(* IEC 61131-3 sources: AXOpen/src/data/app/src/Examples, 4 files *)

(* ---- AxoDataDistributedExample.st ---- *)
USING AXOpen.Core;
USING AXOpen.Data;

NAMESPACE AxoDataDistributedExample

    //<ContextDeclaration>
    {S7.extern=ReadWrite}
    CLASS PUBLIC Context EXTENDS AXOpen.Core.AxoContext
        VAR PUBLIC
            //Controlled unit that needs to manipulate with data
            {#ix-set:AttributeName = "Unit 1"}
            ControlledUnit_1 : ControlledUnit;

            {#ix-set:AttributeName = "Unit 2"}
            ControlledUnit_2 : ControlledUnit;
        END_VAR

        METHOD OVERRIDE Main
            THIS.InitializeRootObject(ControlledUnit);
            ControlledUnit.Run();// run logic of controlled unit
        END_METHOD
    END_CLASS
    //</ContextDeclaration>

    {S7.extern=ReadWrite}
    CLASS PUBLIC SharedHeader_Manager
        EXTENDS AXOpen.Data.AxoDataExchange
        VAR PUBLIC
            {#ix-generic:TOnline}
            {#ix-generic:TPlain as POCO}
            {#ix-attr:[AXOpen.Data.AxoDataEntityAttribute]}
            {#ix-attr:[Container(Layout.Stack)]}
            {#ix-set:AttributeName = "Shared Header"}
            Set : SharedHeader_Data;
        END_VAR
    END_CLASS

    {S7.extern=ReadWrite}
    CLASS PUBLIC SharedHeader_Data
        EXTENDS AXOpen.Data.AxoDataEntity
        VAR PUBLIC
            HeaderPartialName : STRING;
            HeaderIndex : INT;
            HeaderGlogalPass : BOOL;
        END_VAR
    END_CLASS

    {S7.extern=ReadWrite}
    CLASS PUBLIC StationData_Manager
        EXTENDS AXOpen.Data.AxoDataExchange
        VAR PUBLIC
            {#ix-generic:TOnline}
            {#ix-generic:TPlain as POCO}
            {#ix-attr:[AXOpen.Data.AxoDataEntityAttribute]}
            {#ix-attr:[Container(Layout.Stack)]}
            {#ix-set:AttributeName = "Station"}
            Set : Station_Data;
        END_VAR
    END_CLASS

    {S7.extern=ReadWrite}
    CLASS PUBLIC Station_Data EXTENDS AXOpen.Data.AxoDataEntity
        VAR PUBLIC
            StationName : STRING;
            StaionOperation : INT;
            StationPass : BOOL;
        END_VAR
    END_CLASS

     {S7.extern=ReadWrite}
     CLASS PUBLIC ManagerUsage
        VAR PUBLIC
            _id : STRING;
            _create : BOOL;
            _update : BOOL;
            _read : BOOL;
            _delete : BOOL;
        END_VAR

        METHOD PUBLIC Use
            VAR_IN_OUT
                DataManager : AXOpen.Data.AxoDataExchange;
            END_VAR
            IF(_create) THEN
                IF(DataManager.Create(_id).IsDone()) THEN
                    _create := FALSE;
                END_IF;
            END_IF;

            IF(_read) THEN
                IF(DataManager.Read(_id).IsDone()) THEN
                    _read := FALSE;
                END_IF;
            END_IF;

            IF(_update) THEN
                IF(DataManager.Update(_id).IsDone()) THEN
                    _update := FALSE;
                END_IF;
            END_IF;

            IF(_delete) THEN
                IF(DataManager.Delete(_id).IsDone()) THEN
                    _delete := FALSE;
                END_IF;
            END_IF;
        END_METHOD
    END_CLASS

    {S7.extern=ReadWrite}
    CLASS PUBLIC ControlledUnit EXTENDS AXOpen.Core.AxoObject
        VAR PUBLIC

            //<UseDistributedDataAttribute>
            {#ix-attr:[AXOpen.Data.DistributedDataAttribute("default", "headers")]}
            EntityHeader : SharedHeader_Manager;
            {#ix-attr:[AXOpen.Data.DistributedDataAttribute("default", "headers")]}
            ProcessData : StationData_Manager;
            //</UseDistributedDataAttribute>

            HeaderUsage : ManagerUsage;
            ProcessUsage : ManagerUsage;

            //Automatic sequence. Contains logic for automatic operations of this unit.
            AutomatSequence : AutomatSequence;
        END_VAR

        METHOD PUBLIC Run
            SUPER.Run(THIS); //??
            THIS.EntityHeader.Run(THIS)
            THIS.ProcessData.Run(THIS)

            HeaderUsage.Run(THIS);
            ProcessUsage.Run(THIS);

            THIS.Execute();
        END_METHOD

        METHOD PRIVATE Execute
            ProcessData^.Run(THIS); // cyclic call of AxoProcessDataManager
            AutomatSequence.Run(THIS, ^ProcessData);
        END_METHOD
    END_CLASS

    //<Run>
    {S7.extern=ReadWrite}
    CLASS PUBLIC AutomatSequence EXTENDS AXOpen.Core.AxoSequencerContainer
        VAR PRIVATE
            // private reference is used in Main()
            HeaderData : REF_TO SharedHeader_Manager;
            ProcessData : REF_TO StationData_Manager;
        END_VAR

        METHOD INTERNAL Run
            VAR_INPUT
                _parent : IAxoObject;
                _processData : REF_TO StationData_Manager;
                _headerData : REF_TO SharedHeader_Manager;
            END_VAR

            ProcessData := _processData;
            HeaderData := _headerData;
        END_METHOD

        METHOD OVERRIDE Main
            ;//cyclic logic
        END_METHOD
    END_CLASS
    //</Run>

END_NAMESPACE

(* ---- AxoDataExchangeExample.st ---- *)
USING AXOpen.Core;
USING AXOpen;
using AXOpen.Data;

NAMESPACE AxoDataExchangeExample

    //<ContextDeclaration>
    {S7.extern=ReadWrite}
    CLASS PUBLIC Context EXTENDS AXOpen.Core.AxoContext
        VAR PUBLIC
            //Controlled unit that needs to manipulate with data
            ControlledUnit : ControlledUnit;
            //DataManager instance
            DataManager  : AxoProcessDataManager;

            //Testing usage of the manager
            ManagerUsage : ManagerUsage;
        END_VAR

        METHOD OVERRIDE Main

            // DataManager.Run(THIS); - is called iside of controlle unit
            THIS.InitializeRootObject(ControlledUnit);
            ControlledUnit.ProcessData := REF(DataManager);//Set REF to DataManager (reason depth of data structure)
            ControlledUnit.Run();// run logic of controlled unit

            ManagerUsage.Use(DataManager);
        END_METHOD
    END_CLASS
    //</ContextDeclaration>

    //<AxoProcessDataManagerDeclaration>
    {S7.extern=ReadWrite}
    CLASS PUBLIC AxoProcessDataManager EXTENDS AXOpen.Data.AxoDataExchange
        VAR PUBLIC
            {#ix-generic:TOnline}
            {#ix-generic:TPlain as POCO}
            {#ix-attr:[AXOpen.Data.AxoDataEntityAttribute]}
            Set : AxoProcessData; // <- Manager will operate on this member.
        END_VAR
    END_CLASS
    //</AxoProcessDataManagerDeclaration>

    //<AxoProcessDataDeclaration>
    {S7.extern=ReadWrite}
    CLASS PUBLIC AxoProcessData EXTENDS AXOpen.Data.AxoDataEntity
        VAR PUBLIC
            {#ix-set:AttributeName = "Some string"}
            SomeString : STRING;
            {#ix-set:AttributeName = "Some int"}
            SomeInt : INT;

            AllPrimitives : BasePrimitives;
        END_VAR
    END_CLASS
    //</AxoProcessDataDeclaration>

    //<Usage>
    {S7.extern=ReadWrite}
    CLASS PUBLIC ManagerUsage
        VAR PUBLIC
            _id : STRING;
            _create : BOOL;
            _update : BOOL;
            _read : BOOL;
            _delete : BOOL;
        END_VAR

        METHOD PUBLIC Use
            VAR_IN_OUT
                DataManager : AxoProcessDataManager;
            END_VAR
            IF(_create) THEN
                IF(DataManager.Create(_id).IsDone()) THEN
                    _create := FALSE;
                END_IF;
            END_IF;

            IF(_read) THEN
                IF(DataManager.Read(_id).IsDone()) THEN
                    _read := FALSE;
                END_IF;
            END_IF;

            IF(_update) THEN
                IF(DataManager.Update(_id).IsDone()) THEN
                    _update := FALSE;
                END_IF;
            END_IF;

            IF(_delete) THEN
                IF(DataManager.Delete(_id).IsDone()) THEN
                    _delete := FALSE;
                END_IF;
            END_IF;
        END_METHOD
    END_CLASS
    //</Usage>

    //<Execute>
    {S7.extern=ReadWrite}
    CLASS PUBLIC ControlledUnit EXTENDS AXOpen.Core.AxoObject
        VAR PUBLIC
            //Reference to ProcessDataManager
            ProcessData : REF_TO AxoProcessDataManager;
            //Automatic sequence. Contains logic for automatic operations of this unit.
            AutomatSequence : AutomatSequence;
        END_VAR

        METHOD PUBLIC Run
            SUPER.Run(THIS); //??
            THIS.Execute();
        END_METHOD

        METHOD PRIVATE Execute
            ProcessData^.Run(THIS); // cyclic call of AxoProcessDataManager
            AutomatSequence.Run(THIS, ProcessData);
        END_METHOD
    END_CLASS
    //</Execute>

    //<Run>
    {S7.extern=ReadWrite}
    CLASS PUBLIC AutomatSequence EXTENDS AXOpen.Core.AxoSequencerContainer
        VAR PRIVATE
            // private reference is used in Main()
            ProcessData : REF_TO AxoProcessDataManager;
        END_VAR

        METHOD INTERNAL Run
            VAR_INPUT
                _parent : IAxoObject;
                _processData : REF_TO AxoProcessDataManager;
            END_VAR

            ProcessData := _processData;
        END_METHOD

        METHOD OVERRIDE Main
            ;//cyclic logic
        END_METHOD
    END_CLASS
    //</Run>

    {S7.extern=ReadWrite}
    CLASS PUBLIC BasePrimitives //27 vars
        VAR PUBLIC
            vBOOL           :       BOOL	      ;
            vBYTE           :       BYTE	      ;
            vWORD           :       WORD	      ;
            vDWORD          :       DWORD	      ;
            vLWORD	        :       LWORD	      ;
            vSINT           :       SINT	      ;
            vINT	        :       INT           ;
            vDINT	        :       DINT	      ;
            vLINT	        :       LINT	      ;
            vUSINT	        :       USINT	      ;
            vUINT	        :       UINT	      ;
            vUDINT	        :       UDINT	      ;
            vULINT	        :       ULINT	      ;
            vREAL	        :       REAL	      ;
            vLREAL	        :       LREAL	      ;
            vTIME	        :       TIME	      ;
            vLTIME	        :       LTIME	      ;
            vDATE	        :       DATE	      ;
            vLDATE	        :       LDATE	      ;
            vTIME_OF_DAY	:       TIME_OF_DAY   ;
            vLTIME_OF_DAY	:       LTIME_OF_DAY  ;
            vDATE_AND_TIME  :      DATE_AND_TIME  ;
            vLDATE_AND_TIME :      LDATE_AND_TIME ;
            vCHAR	        :       CHAR	      ;
            vWCHAR	        :       WCHAR	      ;
            vSTRING         :       STRING	      ;
            vWSTRING        :       WSTRING	      ;
        END_VAR
    END_CLASS

END_NAMESPACE

(* ---- AxoDataFragmentExchangeExample.st ---- *)
USING AXOpen.Core;
USING AXOpen.Data;

NAMESPACE AxoDataFramentsExchangeExample

    //<ContextDeclaration>
    {S7.extern=ReadWrite}
    CLASS PUBLIC Context EXTENDS AXOpen.Core.AxoContext
        VAR PUBLIC
            //Controlled unit that needs to manipulate with data
            ControlledUnit : ControlledUnit;
            //DataManager instance
            DataManager  : AxoProcessDataManager;

            //Testing usage of the manager
            ManagerUsage : ManagerUsage;
        END_VAR

        METHOD OVERRIDE Main

            // DataManager.Run(THIS); - is called iside of controlle unit
            ControlledUnit.ProcessData := REF(DataManager);//Set REF to DataManager (reason depth of data structure)
            ControlledUnit.Run(THIS);// run logic of controlled unit

            ManagerUsage.Use(DataManager);
        END_METHOD
    END_CLASS
    //</ContextDeclaration>

    //<AxoProcessDataManagerDeclaration>
    {S7.extern=ReadWrite}
    CLASS PUBLIC AxoProcessDataManager
        EXTENDS AXOpen.Data.AxoDataFragmentExchange
        VAR PUBLIC
            {#ix-attr:[AXOpen.Data.AxoDataFragmentAttribute]}
            SharedHeader : SharedDataHeaderManager;
            {#ix-attr:[AXOpen.Data.AxoDataFragmentAttribute]}
            Station_1 : Station_1_ProcessDataManager;
        END_VAR
    END_CLASS
    //</AxoProcessDataManagerDeclaration>

    {S7.extern=ReadWrite}
    CLASS PUBLIC SharedDataHeaderManager
        EXTENDS AXOpen.Data.AxoDataExchange
        VAR PUBLIC
            {#ix-generic:TOnline}
            {#ix-generic:TPlain as POCO}
            {#ix-attr:[AXOpen.Data.AxoDataEntityAttribute]}
            {#ix-attr:[Container(Layout.Stack)]}
            {#ix-set:AttributeName = "Shared Header"}
            Set : SharedDataHeaderData;
        END_VAR
    END_CLASS

    {S7.extern=ReadWrite}
    CLASS PUBLIC SharedDataHeaderData
        EXTENDS AXOpen.Data.AxoDataEntity
        VAR PUBLIC
            {#ix-set:AttributeName = "Some string"}
            SomeString : STRING;
            {#ix-set:AttributeName = "Some int"}
            SomeInt : INT;
            {#ix-set:AttributeName = "Some bool"}
            SomeBool : BOOL;
        END_VAR
    END_CLASS

    {S7.extern=ReadWrite}
    CLASS PUBLIC Station_1_ProcessDataManager
        EXTENDS AXOpen.Data.AxoDataExchange
        VAR PUBLIC
            {#ix-generic:TOnline}
            {#ix-generic:TPlain as POCO}
            {#ix-attr:[AXOpen.Data.AxoDataEntityAttribute]}
            {#ix-attr:[Container(Layout.Stack)]}
            {#ix-set:AttributeName = "Station 1"}
            Set : Station_1_Data;
        END_VAR
    END_CLASS

    {S7.extern=ReadWrite}
    CLASS PUBLIC Station_1_Data EXTENDS AXOpen.Data.AxoDataEntity
        VAR PUBLIC
            {#ix-set:AttributeName = "Some string st"}
            SomeString : STRING;
            {#ix-set:AttributeName = "Some int st"}
            SomeInt : INT;
            {#ix-set:AttributeName = "Some bool st"}
            SomeBool : BOOL;
        END_VAR
    END_CLASS

     //<Usage>
     {S7.extern=ReadWrite}
     CLASS PUBLIC ManagerUsage
        VAR PUBLIC
            _id : STRING;
            _create : BOOL;
            _update : BOOL;
            _read : BOOL;
            _delete : BOOL;
        END_VAR

        METHOD PUBLIC Use
            VAR_IN_OUT
                DataManager : AxoProcessDataManager;
            END_VAR
            IF(_create) THEN
                IF(DataManager.Create(_id).IsDone()) THEN
                    _create := FALSE;
                END_IF;
            END_IF;

            IF(_read) THEN
                IF(DataManager.Read(_id).IsDone()) THEN
                    _read := FALSE;
                END_IF;
            END_IF;

            IF(_update) THEN
                IF(DataManager.Update(_id).IsDone()) THEN
                    _update := FALSE;
                END_IF;
            END_IF;

            IF(_delete) THEN
                IF(DataManager.Delete(_id).IsDone()) THEN
                    _delete := FALSE;
                END_IF;
            END_IF;
        END_METHOD
    END_CLASS
    //</Usage>

    //<Execute>
    {S7.extern=ReadWrite}
    CLASS PUBLIC ControlledUnit EXTENDS AXOpen.Core.AxoObject
        VAR PUBLIC
            //Reference to ProcessDataManager
            ProcessData : REF_TO AxoProcessDataManager;
            //Automatic sequence. Contains logic for automatic operations of this unit.
            AutomatSequence : AutomatSequence;
        END_VAR

        METHOD PUBLIC Run
            VAR_INPUT
                _parent : IAxoContext;
            END_VAR
            THIS.Initialize(_parent);
            THIS.Execute();
        END_METHOD

        METHOD PRIVATE Execute
            ProcessData^.Run(THIS); // cyclic call of AxoProcessDataManager
            AutomatSequence.Run(THIS, ProcessData);
        END_METHOD
    END_CLASS
    //</Execute>

    //<Run>
    {S7.extern=ReadWrite}
    CLASS PUBLIC AutomatSequence EXTENDS AXOpen.Core.AxoSequencerContainer
        VAR PRIVATE
            // private reference is used in Main()
            ProcessData : REF_TO AxoProcessDataManager;
        END_VAR

        METHOD INTERNAL Run
            VAR_INPUT
                _parent : IAxoObject;
                _processData : REF_TO AxoProcessDataManager;
            END_VAR

            ProcessData := _processData;
        END_METHOD

        METHOD OVERRIDE Main
            ;//cyclic logic
        END_METHOD
    END_CLASS
    //</Run>

END_NAMESPACE

(* ---- AxoDataPersistentExchangeExample.st ---- *)
USING AXOpen.Core;
USING AXOpen;
using AXOpen.Data;

NAMESPACE AxoDataPersistentExchangeExample

    //<ContextDeclaration>
    {S7.extern=ReadWrite}
    CLASS PUBLIC Context EXTENDS AXOpen.Core.AxoContext
        VAR PUBLIC
            //persistent manager instance
            DataManager : AXOpen.Data.AxoDataPersistentExchange;
            //Testing usage of the manager
            ManagerUsage : ManagerUsage;
            // Object that propertie will be tracked by persistent manager
            PersistentRootObject : PersistentRootObject;
            _rootObject :   AxoObject;
        END_VAR

        METHOD OVERRIDE Main
            _rootObject.InitializeWithContext(THIS);
            DataManager.Run(_rootObject);
            ManagerUsage.Use(DataManager);
        END_METHOD
    END_CLASS
    //</ContextDeclaration>

    //<Usage>
    {S7.extern=ReadWrite}
    CLASS PUBLIC ManagerUsage EXTENDS AxOpen.Core.AxoObject
        VAR PUBLIC
            _persistentGroupId : STRING;
            _update : BOOL;
            _read : BOOL;
            _updateAll : BOOL;
            _readAll : BOOL;
            _exist : BOOL;
            _recordExist : BOOL;
        END_VAR

        METHOD PUBLIC Use
            VAR_IN_OUT
                DataManager : AXOpen.Data.AxoDataPersistentExchange;
            END_VAR

            IF(_read) THEN
                IF(DataManager.InvokeRead(THIS,_persistentGroupId)) THEN
                    ;
                END_IF;

                IF(DataManager.IsReadDone(THIS)) THEN
                    _read := FALSE;
                END_IF;
            END_IF;

            IF(_update) THEN
                IF(DataManager.InvokeUpdate(THIS,_persistentGroupId)) THEN
                   ;
                END_IF;

                IF(DataManager.IsUpdateDone(THIS)) THEN
                    _update := FALSE;
                END_IF;
            END_IF;

            IF(_readAll) THEN
                IF(DataManager.InvokeReadAll(THIS)) THEN
                   ;
                END_IF;
                IF(DataManager.IsReadAllDone(THIS)) THEN
                    _readAll := FALSE;
                END_IF;
            END_IF;

            IF(_updateAll) THEN
                IF(DataManager.InvokeUpdateAll(THIS)) THEN
                    ;
                END_IF;

                IF(DataManager.IsUpdateAllDone(THIS)) THEN
                    _updateAll := FALSE;
                END_IF;
            END_IF;

            IF(_exist) THEN
                IF(DataManager.InvokeEntityExist(THIS, _persistentGroupId)) THEN
                    ;
                END_IF;

                IF(DataManager.IsEntityExistDone(THIS)) THEN
                    _exist := FALSE;
                    _recordExist := DataManager.Operation._exist;
                END_IF;
            END_IF;
        END_METHOD
    END_CLASS
    //</ConcurrentUsage>

    //<PersistentAttribute>
    {S7.extern=ReadWrite}
    CLASS PUBLIC PersistentRootObject
        VAR PUBLIC
            NotPersistentVariable : BOOL;

            {#ix-attr:[Persistent()]}
            {#ix-set:AttributeName = "PersistentVariable_1 (in default pg.))"}
            PersistentVariable_1 : INT; // will be saved to 'default' persistent group

            {#ix-attr:[Persistent("default","1")]} // will be saved to 'default' and '1' persistent group
            {#ix-set:AttributeName = "PersistentVariable_2 (in default & 1 pg.)"}
            PersistentVariable_2 : INT;

            {#ix-attr:[Container(Layout.Stack)]}
            {#ix-attr:[Group(GroupLayout.GroupBox)]}
            {#ix-set:AttributeName = "PropertyWithPersistentMember"}
            PropertyWithPersistentMember : ObjectWithPersistentMember;
        END_VAR
    END_CLASS

    {S7.extern=ReadWrite}
    CLASS PUBLIC ObjectWithPersistentMember
        VAR PUBLIC
            NotPersistentVariable : INT;

            {#ix-attr:[Persistent("2")]}
            {#ix-attr:[Container(Layout.Stack)]}
            {#ix-attr:[Group(GroupLayout.GroupBox)]}
            {#ix-set:AttributeName = "InitializedPrimitives (in 2 pg.)"}
            InitializedPrimitives : InitializedPrimitives;
        END_VAR
    END_CLASS

    {S7.extern=ReadWrite}
    CLASS PUBLIC InitializedPrimitives
        VAR PUBLIC
            myBOOL          :       BOOL	      := true;
            myBYTE          :       BYTE	      := BYTE#255;
            myWORD          :       WORD	      := WORD#60000;
            myDWORD         :       DWORD	      := DWORD#16#ABCD_EF01;
            myLWORD	        :       LWORD	      := LWORD#18446744073709551615;
            mySINTMin       :       SINT	      := SINT#-128;
            mySINTMax       :       SINT	      := SINT#127;
            myINT	        :       INT           := INT#32767;
            myDINT	        :       DINT	      := DINT#2147483647;
            myLINT	        :       LINT	      := LINT#9223372036854775807;
            myUSINT	        :       USINT	      := USINT#255;
            myUINT	        :       UINT	      := UINT#65535;
            myUDINT	        :       UDINT	      := UDINT#4294967295;
            myULINT	        :       ULINT	      := ULINT#18446744073709551615;
            myREAL	        :       REAL	      := REAL#+3.402823e+38;
            myLREAL	        :       LREAL	      := LREAL#1.79769313486231e+308;
            myTIME	        :       TIME	      := TIME#2147483647ms;
            myLTIME	        :       LTIME	      := LTIME#100000d2h4m8s16ms32ns;
            myDATE	        :       DATE	      := DATE#2262-04-11;
            myLDATE	        :       LDATE	      := LDATE#2262-04-11;
            myTIME_OF_DAY	:       TIME_OF_DAY   := TIME_OF_DAY#23:59:59.999999999;
            myLTIME_OF_DAY	:       LTIME_OF_DAY  := LTIME_OF_DAY#23:59:59.999999999;
            myDATE_AND_TIME :      DATE_AND_TIME  := DATE_AND_TIME#2262-04-11-23:47:16.854775807;
            myLDATE_AND_TIME :      LDATE_AND_TIME := LDATE_AND_TIME#2262-04-11-23:47:16.854775807;
            myCHAR	        :       CHAR	      := CHAR#255;
            myWCHAR	        :       WCHAR	      := WCHAR#65535;
            mySTRING        :       STRING	      := 'o\zxcvbnm,./asdfghjkl;\\qwertyuiop[]1234567890-~!@#^&*()_+';
            myWSTRING       :       WSTRING	      := WSTRING#"o\zxcvbnm,./asdfghjkl;'\qwertyuiop[]1234567890-~!@#^&*()_+";
        END_VAR
    END_CLASS
    //</PersistentAttribute>

END_NAMESPACE
